FUNCTION_BLOCK CLOCK (* Clock signal generator *)
  (* Standard: 61499-2 *)
  (* Version 1.0, 2008-11-09, Cheng Pang, The University of Auckland, Stable build. *)
  (* Compiler header: package fb.rt.pnp; *)
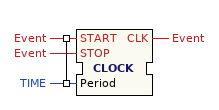
  EVENT_INPUT
    START WITH Period;
    STOP;
  END_EVENT
  EVENT_OUTPUT
    CLK;
  END_EVENT
  VAR_INPUT
    Period : TIME;
  END_VAR
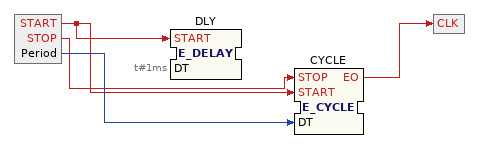
  FBS
    DLY : E_DELAY(DT := t#1ms);
    CYCLE : E_CYCLE;
  END_FBS
  EVENT_CONNECTIONS
    START TO DLY.START;
    STOP TO CYCLE.STOP;
    START TO CYCLE.START;
    CYCLE.EO TO CLK;
  END_CONNECTIONS
  DATA_CONNECTIONS
    Period TO CYCLE.DT;
  END_CONNECTIONS
END_FUNCTION_BLOCK
